TYPE eUnit :
(
    mm  := 0,
    m   := 1,
    deg := 2,
    rad := 3
);
END_TYPE

(* stored: Version 1.1.0.1, ProductVersion 3.1.4026.18
   DUT eUnit: Id {a8e5f521-c1b2-4a73-87a0-100000000001} *)
